Yaskawa INFORM job: u_tempsTRJ0.JBI

/JOB
//NAME u_tempsTRJ0
///FOLDERNAME DEMO
//POS
///NPOS 21,0,21,0,0,0
///USER 2
///TOOL 7
///POSTYPE USER
///RECTAN
///RCONF 1,0,0,0,0,0,0,0,0,0,0,0,0,0,0,0,0,0,0,0,0,0,0,0
C00000=0.000,0.000,0.000,-180.0000,-0.0000,-90.0000
C00001=0.000,0.000,200.000,-180.0000,-0.0000,-90.0000
C00002=0.000,0.000,0.000,-180.0000,-0.0000,-90.0000
C00003=0.000,0.000,200.000,-180.0000,-0.0000,-90.0000
C00004=0.000,0.000,0.000,-180.0000,-0.0000,-90.0000
C00005=0.000,0.000,200.000,-180.0000,-0.0000,-90.0000
C00006=0.000,0.000,0.000,-180.0000,-0.0000,-90.0000
C00007=0.000,0.000,200.000,-180.0000,-0.0000,-90.0000
C00008=0.000,0.000,0.000,-180.0000,-0.0000,-90.0000
C00009=0.000,0.000,200.000,-180.0000,-0.0000,-90.0000
C00010=0.000,0.000,0.000,-180.0000,-0.0000,-90.0000
C00011=0.000,0.000,200.000,-180.0000,-0.0000,-90.0000
C00012=0.000,0.000,0.000,-180.0000,-0.0000,-90.0000
C00013=0.000,0.000,200.000,-180.0000,-0.0000,-90.0000
C00014=0.000,0.000,0.000,-180.0000,-0.0000,-90.0000
C00015=0.000,0.000,200.000,-180.0000,-0.0000,-90.0000
C00016=0.000,0.000,0.000,-180.0000,-0.0000,-90.0000
C00017=0.000,0.000,200.000,-180.0000,-0.0000,-90.0000
C00018=0.000,0.000,0.000,-180.0000,-0.0000,-90.0000
C00019=0.000,0.000,200.000,-180.0000,-0.0000,-90.0000
C00020=0.000,0.000,0.000,-180.0000,-0.0000,-90.0000
///TOOL 0
///POSTYPE ANGLE
///ANGLE
EC00000=-0.0000,90.0000
EC00001=-0.0000,90.0000
EC00002=-0.0000,90.0000
EC00003=-0.0000,90.0000
EC00004=-0.0000,90.0000
EC00005=-0.0000,90.0000
EC00006=-0.0000,90.0000
EC00007=-0.0000,90.0000
EC00008=-0.0000,90.0000
EC00009=-0.0000,90.0000
EC00010=-0.0000,90.0000
EC00011=-0.0000,90.0000
EC00012=-0.0000,90.0000
EC00013=-0.0000,90.0000
EC00014=-0.0000,90.0000
EC00015=-0.0000,90.0000
EC00016=-0.0000,90.0000
EC00017=-0.0000,90.0000
EC00018=-0.0000,90.0000
EC00019=-0.0000,90.0000
EC00020=-0.0000,90.0000
//INST
///DATE 2021/09/28 14:58
///COMM
///ATTR SC,RW,RJ
////FRAME USER 2
///GROUP1 RB1
///GROUP2 ST1
NOP
SPEED V=10.0
SMOVL C00000 +MOVJ EC00000
SMOVL C00001 +MOVJ EC00001
SMOVL C00002 +MOVJ EC00002
SMOVL C00003 +MOVJ EC00003
SMOVL C00004 +MOVJ EC00004
SMOVL C00005 +MOVJ EC00005
SMOVL C00006 +MOVJ EC00006
SMOVL C00007 +MOVJ EC00007
SMOVL C00008 +MOVJ EC00008
SMOVL C00009 +MOVJ EC00009
SMOVL C00010 +MOVJ EC00010
SMOVL C00011 +MOVJ EC00011
SMOVL C00012 +MOVJ EC00012
SMOVL C00013 +MOVJ EC00013
SMOVL C00014 +MOVJ EC00014
SMOVL C00015 +MOVJ EC00015
SMOVL C00016 +MOVJ EC00016
SMOVL C00017 +MOVJ EC00017
SMOVL C00018 +MOVJ EC00018
SMOVL C00019 +MOVJ EC00019
SMOVL C00020 +MOVJ EC00020
END
